// SIMATIC S7-200 project (STEP 7-Micro/WIN), CPU 224XP REL 02.01

SYMBOL_TABLE USER1
send_enable      V1020.0
gps_lat_deg      VW50
gps_lat_min      VD52
gps_lat_dir      VB56
gps_long_deg     VW57
gps_long_min     VD59
gps_long_dir     VB64
gps_alt          VD65
gps_alt_u        VB69
gps_speed        VD70
msg_value        VB1990
msg              VB2000
counter          C0
counter_delay    VW102
counter_send     V10.0
counter_max      VW104
counter_stop     V10.1
table            VW2500
table_count      VW2502
table_out        VW110
table_out_s      VB112
init_pin         VB1001
init_srv         VB1006
init_busy        V1000.0
init_done        V1000.1
init_ab          V1000.2
init_st          VW1026
send_ready       V1100.3
send_to          VB1050
send_busy        V1100.0
send_done        V1100.1
send_ab          V1100.2
send_st          VW1126
send_en          V1100.4
send_stop        V1100.5
rcv_busy         V1200.0
rcv_done         V1200.1
rcv_ab           V1200.2
rcv_buf          VB1210
rcv_msg          VB1238
rcv_st           VW1250
END_SYMBOL_TABLE

ORGANIZATION_BLOCK MAIN:OB1
TITLE=PROGRAM COMMENTS
BEGIN
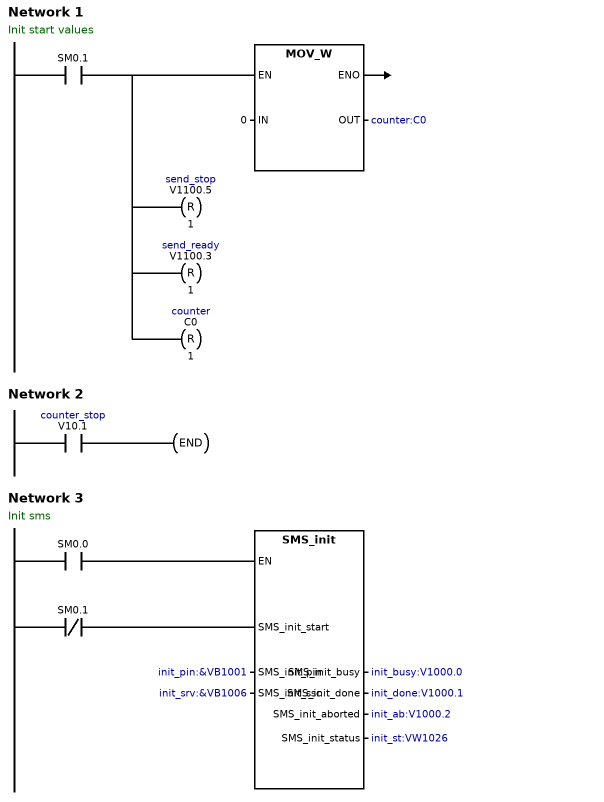
Network 1
// Init start values
LD     SM0.1
MOVW   0, counter:C0
R      send_stop:V1100.5, 1
R      send_ready:V1100.3, 1
R      counter:C0, 1
Network 2
LD     counter_stop:V10.1
END
Network 3
// Init sms
LD     SM0.0
=      L60.0
LDN    SM0.1
=      L63.7
LD     L60.0
CALL   SMS_init:SBR2, L63.7, &init_pin:VB1001, &init_srv:VB1006, init_busy:V1000.0, init_done:V1000.1, init_ab:V1000.2, init_st:VW1026
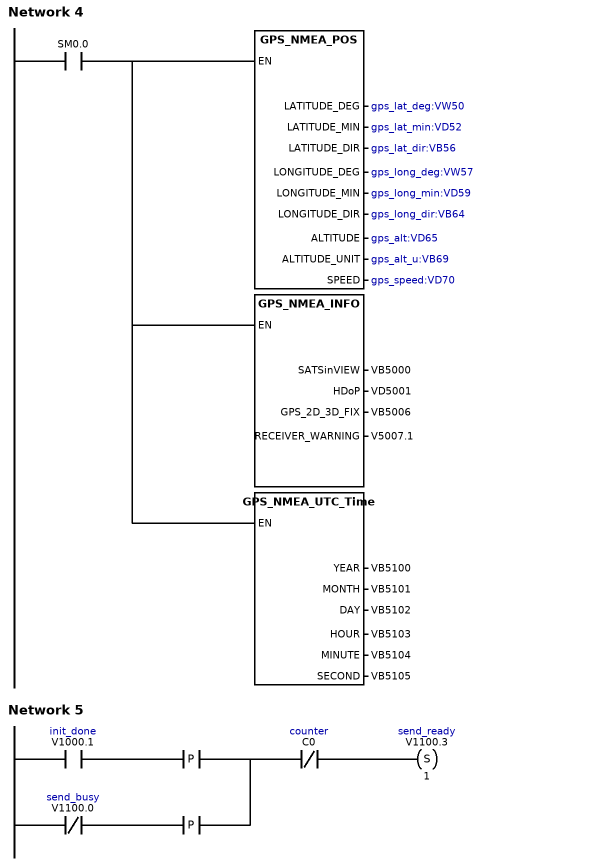
Network 4
LD     SM0.0
CALL   GPS_NMEA_POS:SBR6, gps_lat_deg:VW50, gps_lat_min:VD52, gps_lat_dir:VB56, gps_long_deg:VW57, gps_long_min:VD59, gps_long_dir:VB64, gps_alt:VD65, gps_alt_u:VB69, gps_speed:VD70
CALL   GPS_NMEA_INFO:SBR7, VB5000, VD5001, VB5006, V5007.1
CALL   GPS_NMEA_UTC_Time:SBR8, VB5100, VB5101, VB5102, VB5103, VB5104, VB5105
Network 5
LD     init_done:V1000.1
EU
LDN    send_busy:V1100.0
EU
OLD
AN     counter:C0
S      send_ready:V1100.3, 1
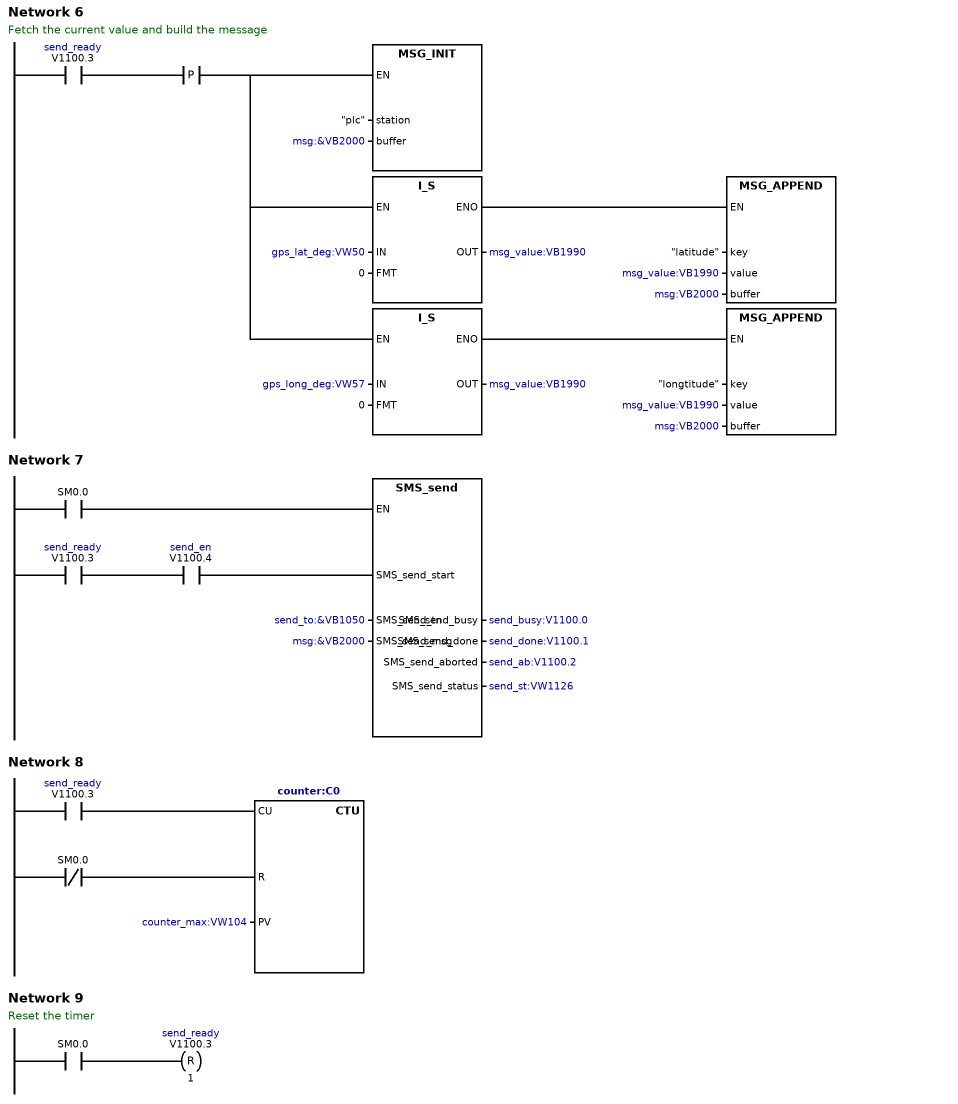
Network 6
// Fetch the current value and build the message
LD     send_ready:V1100.3
EU
LPS
CALL   MSG_INIT:SBR0, "plc", &msg:VB2000
ITS    gps_lat_deg:VW50, msg_value:VB1990, 0
AENO
CALL   MSG_APPEND:SBR5, "latitude", msg_value:VB1990, msg:VB2000
LPP
ITS    gps_long_deg:VW57, msg_value:VB1990, 0
AENO
CALL   MSG_APPEND:SBR5, "longtitude", msg_value:VB1990, msg:VB2000
Network 7
LD     SM0.0
=      L60.0
LD     send_ready:V1100.3
A      send_en:V1100.4
=      L63.7
LD     L60.0
CALL   SMS_send:SBR3, L63.7, &send_to:VB1050, &msg:VB2000, send_busy:V1100.0, send_done:V1100.1, send_ab:V1100.2, send_st:VW1126
Network 8
LD     send_ready:V1100.3
LDN    SM0.0
CTU    counter:C0, counter_max:VW104
Network 9
// Reset the timer
LD     SM0.0
R      send_ready:V1100.3, 1
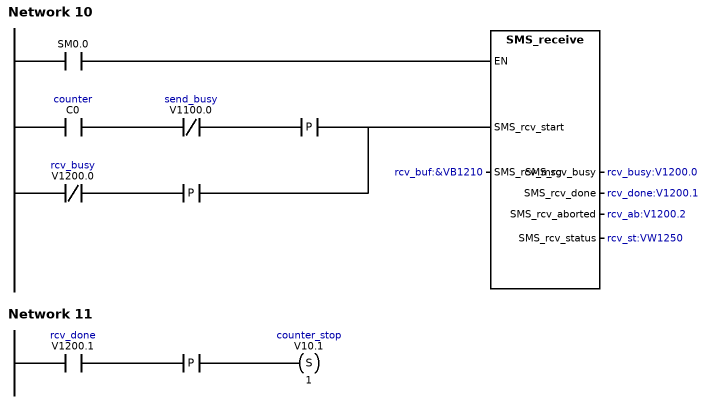
Network 10
LD     SM0.0
=      L60.0
LD     counter:C0
AN     send_busy:V1100.0
EU
LDN    rcv_busy:V1200.0
EU
OLD
=      L63.7
LD     L60.0
CALL   SMS_receive:SBR4, L63.7, &rcv_buf:VB1210, rcv_busy:V1200.0, rcv_done:V1200.1, rcv_ab:V1200.2, rcv_st:VW1250
Network 11
LD     rcv_done:V1200.1
EU
S      counter_stop:V10.1, 1
END_ORGANIZATION_BLOCK

SUBROUTINE_BLOCK MSG_INIT:SBR0
TITLE=SUBROUTINE COMMENTS
VAR_INPUT
station:?;	// LD0 
buffer:DWORD;	// LD4 
END_VAR
VAR
year:BYTE;	// LB8 
month:BYTE;	// LB9 
day:BYTE;	// LB10 
hour:BYTE;	// LB11 
minute:BYTE;	// LB12 
seconds:BYTE;	// LB13 
tmp:INT;	// LW14 
tmp_s:DWORD;	// LD16 
END_VAR
BEGIN
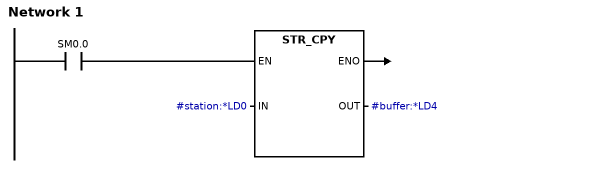
Network 1
LD     SM0.0
SCPY   *#station:LD0, *#buffer:LD4
END_SUBROUTINE_BLOCK

// SBR1: protected block, not included

// SBR2: protected block, not included

// SBR3: protected block, not included

// SBR4: protected block, not included

SUBROUTINE_BLOCK MSG_APPEND:SBR5
TITLE=SUBROUTINE COMMENTS
VAR_INPUT
key:?;	// LD0 
value:?;	// LD4 
buffer:?;	// LD8 
END_VAR
BEGIN
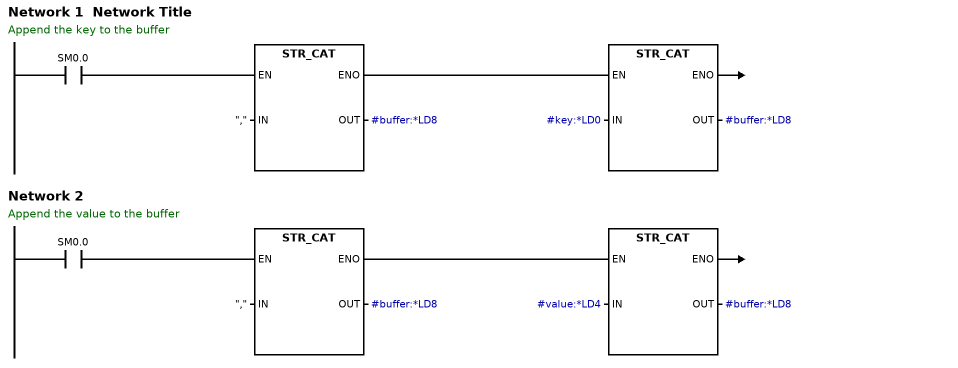
Network 1 // Network Title
// Append the key to the buffer
LD     SM0.0
SCAT   ",", *#buffer:LD8
AENO
SCAT   *#key:LD0, *#buffer:LD8
Network 2
// Append the value to the buffer
LD     SM0.0
SCAT   ",", *#buffer:LD8
AENO
SCAT   *#value:LD4, *#buffer:LD8
END_SUBROUTINE_BLOCK

// SBR6: protected block, not included

// SBR7: protected block, not included

DATA_BLOCK_TAB USER1
BEGIN
//DATA PAGE COMMENTS
//Press F1 for help and example data page
         counter_delay, 40   // counter incrementation delay, s/10
         counter_max, 3      // maximumum counter value
//table:VW2000 +20                   // counter table length
         init_pin, ""
         init_srv, "+37129202020"
         send_to, "+37129252613"
VB1100   2#10000             // enables/disables SMS sending
END_DATA_BLOCK_TAB
